TYPE TcoInsightInspectionControl_v_5_x_x : STRUCT
    EnableResultsBuffering AT %Q* : BOOL;
    AcknowledgeInspectionResults AT %Q* : BOOL;
    ExtendedUserDataSet AT %Q* : BOOL;
    ExecuteCommand AT %Q* : BOOL;
    ClearError AT %Q* : BOOL;
END_STRUCT
END_TYPE

(* stored: Version 1.1.0.1, ProductVersion 3.1.4024.11
   DUT TcoInsightInspectionControl_v_5_x_x: Id {3444326b-467a-0f66-257c-8286be44d747} *)
